Universal Robots PolyScope program: Wheel_holder.urp

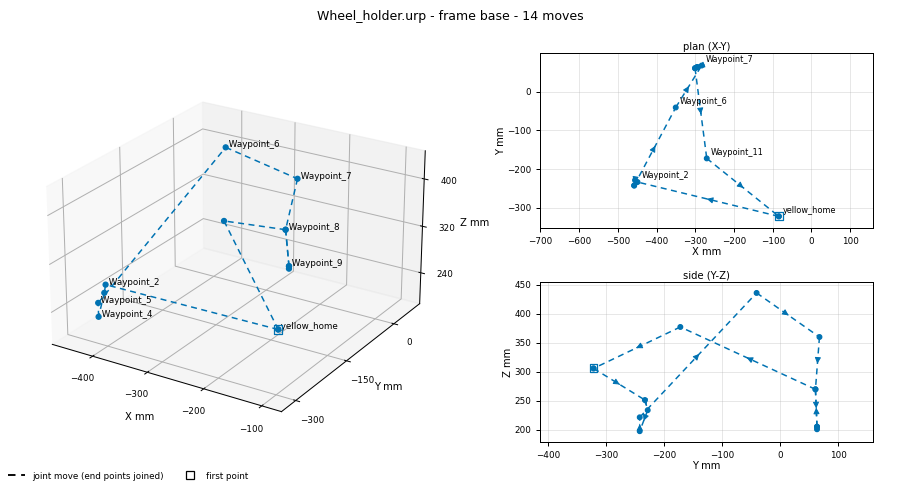
[picture p0: tool path of Wheel_holder.urp in frame base, 14 of 14 moves have a stored position in this frame; points joined in program order, loops and branches not executed]
Program Wheel_holder (installation=default directory=/programs/usbdisk/Zahra1 createdIn=5.11.11.1010533 lastSavedIn=5.11.11.1010533 robotSerialNumber=20205300864)
Calibrated DH parameters: a=[-0.000166, -0.243494, -0.153108, 0.000057, -0.000123, 0]; d=[0.151897, -1.34267, 53.988124, -52.514559, 0.085283, 0.092193]; alpha=[1.572472, -0.003756, 0.002824, 1.570807, -1.572621, 0]; deltaTheta=[0, 0.020704, 7.033215, -0.770746, 0.000004, 0]
Robot Program (runOnlyOnce=true)
  MoveJ speed 60 deg/s, acceleration 80 deg/s^2 (useActiveTCP=true) feature=Base
    Waypoint yellow_home: TCP in base x=-84.299 y=-321.875 z=305.481 mm, rx=-2.0809 ry=-2.2572 rz=0.0984 rad; joints [-79.978, -91.201, -87.971, -91.7, 84.671, 815.506] deg
    Waypoint Waypoint_2: TCP in base x=-449.381 y=-233.265 z=250.97 mm, rx=3.1099 ry=-0.1421 rz=-0.16 rad; joints [-136.989, -138.499, -35.609, -90.672, 86.621, 858.104] deg
    URCap Gripper (Robotiq_Grippers, Robotiq Inc.) dataModel(position=25.098039215686274, force=94.0, speed=40.0, positionInDouble=25.098039215686274, forceInDouble=94.0, speedInDouble=40.0, slaveIds=[9], blocking=true, robotCompliant=false)
    Waypoint Waypoint_3: TCP in base x=-455.729 y=-228.445 z=233.447 mm, rx=3.0708 ry=-0.0583 rz=-0.0252 rad; joints [-138.95, -141.463, -34.006, -91.031, 92.194, 853.304] deg
    Waypoint Waypoint_4: TCP in base x=-457.962 y=-242.224 z=197.193 mm, rx=3.1318 ry=0.0176 rz=-0.0237 rad; joints [-137.479, -145.644, -34.715, -88.521, 89.672, 851.887] deg
    URCap Gripper (Robotiq_Grippers, Robotiq Inc.) dataModel(position=75.68627450980392, force=94.0, speed=40.0, positionInDouble=75.68627450980392, forceInDouble=94.0, speedInDouble=40.0, slaveIds=[9], blocking=true, robotCompliant=false)
    Waypoint Waypoint_5: TCP in base x=-457.953 y=-242.233 z=221.159 mm, rx=3.1318 ry=0.0176 rz=-0.0238 rad; joints [-137.46, -146.242, -27.094, -95.541, 89.656, 851.891] deg
    Waypoint Waypoint_6: TCP in base x=-350.59 y=-40.654 z=435.634 mm, rx=3.1002 ry=0.0439 rz=-0.02 rad; joints [-152.062, -110.196, -27.065, -130.904, 91.596, 836.383] deg
    Waypoint Waypoint_7: TCP in base x=-283.584 y=67.725 z=359.651 mm, rx=-3.1315 ry=-0.0151 rz=-0.0282 rad; joints [-166.712, -83.397, -80.431, -107.198, 89.693, 822.809] deg
    Waypoint Waypoint_8: TCP in base x=-300.723 y=60.827 z=269.441 mm, rx=3.133 ry=0.0152 rz=0.1117 rad; joints [-166.714, -87.226, -100.393, -86.169, 91.34, 822.803] deg
    Waypoint Waypoint_9: TCP in base x=-295.261 y=63.507 z=204.907 mm, rx=3.1314 ry=-0.0044 rz=0.0252 rad; joints [-166.85, -89.764, -117.443, -63.451, 90.842, 823.475] deg
    Waypoint Waypoint_10: TCP in base x=-295.278 y=63.503 z=200.524 mm, rx=3.1313 ry=-0.0045 rz=0.0251 rad; joints [-166.853, -90.312, -118.228, -62.112, 90.846, 823.479] deg
    URCap Gripper (Robotiq_Grippers, Robotiq Inc.) dataModel(position=25.098039215686274, force=94.0, speed=40.0, positionInDouble=25.098039215686274, forceInDouble=94.0, speedInDouble=40.0, slaveIds=[9], blocking=true, robotCompliant=false)
    Waypoint Waypoint_9: TCP in base x=-295.261 y=63.507 z=204.907 mm, rx=3.1314 ry=-0.0044 rz=0.0252 rad; joints [-166.85, -89.764, -117.443, -63.451, 90.842, 823.475] deg
    Waypoint Waypoint_8: TCP in base x=-300.723 y=60.827 z=269.441 mm, rx=3.133 ry=0.0152 rz=0.1117 rad; joints [-166.714, -87.226, -100.393, -86.169, 91.34, 822.803] deg
    Waypoint Waypoint_11: TCP in base x=-270.489 y=-172.183 z=376.926 mm, rx=3.1313 ry=0.1014 rz=-0.0512 rad; joints [-123.078, -90.743, -69.735, -107.96, 88.709, 863.264] deg
    Waypoint yellow_home: TCP in base x=-84.299 y=-321.875 z=305.481 mm, rx=-2.0809 ry=-2.2572 rz=0.0984 rad; joints [-79.978, -91.201, -87.971, -91.7, 84.671, 815.506] deg
